ABB RobotStudio station: GoHolo_Simulation.rspag

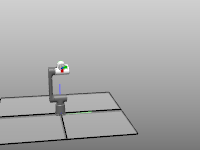
--- station ---
Station GoFa_Simulation (saved by RobotStudio 21.2.9526.0)
Controller GoFa
  mechanical unit ROB_1: CRB15000_5_95__01_2, 6 joints, base frame (0, 0, 0) mm
Layout (positions relative to the parent item):
  - CRB15000_5_95__01_2 [mechanism, from Robots\CRB15000_5_95__01.rslib] at (0, 0, 0) mm; joint values [0, 0, 0, 0, 0, 0] (rad or m)
Targets, tools, work objects and paths stored in the station and not in the controller backup, written as RAPID:
! task T_ROB1
MODULE module_MAIN
  CONST robtarget below:=[[500,0,500],[0,0,0,1],[0,0,0,0],[9E+09,9E+09,9E+09,9E+09,9E+09,9E+09]];
ENDMODULE

! task T_ROB1
MODULE MAINmodul
  PROC goHome()
    MoveJ pHome,v1000,fine,tool0\WObj:=wobj0;
  ENDPROC
ENDMODULE

! task T_ROB1
MODULE module_EGM
  PERS tooldata tEGM:=[TRUE,[[0,0,0],[1,0,0,0]],[0.001,[0,0,0.001],[1,0,0,0],0,0,0]];
  PROC EGM_Setup_UdpUC_Val()
    init_Val;
  ENDPROC
ENDMODULE

! task T_ROB1
MODULE EGM_Guidance
  PERS robtarget Target_10:=[[455.426,100,685.001],[0.5,-0.000000018,0.866025,0.000000059],[0,-1,0,0],[9E+09,9E+09,9E+09,9E+09,9E+09,9E+09]];
  PROC move()
    SingArea \LockAxis4;
  ENDPROC
  PROC EGM_UdpUC_VAL_Tool()
    EGM_Setup_UdpUC_Val;
    move;
    WaitTime 60;
    MoveJ Target_10,v100,fine,tEGM\WObj:=wobj0;
  ENDPROC
ENDMODULE

! task T_ROB1
MODULE module_WIZARD
  PERS robtarget Location3:=[[-0.096782632,525.209777832,576.337219238],[0.606442034,-0.534831524,0.457359105,0.370143116],[-1,-1,1,4],[-170.223126067,9E+09,9E+09,9E+09,9E+09,9E+09]];
  CONST jointtarget j00:=[[0,0,0,0,0,0],[0,0,0,0,0,0]];
  CONST jointtarget j90:=[[90,0,0,0,0,0],[0,0,0,0,0,0]];
  CONST jointtarget j80:=[[0,0,80,0,0,0],[0,0,0,0,0,0]];
  CONST jointtarget j20:=[[20,20,20,20,20,20],[0,0,0,0,0,0]];
  CONST jointtarget j30:=[[30,30,30,30,30,30],[0,0,0,0,0,0]];
  CONST jointtarget j30neg:=[[-30,-30,-30,-30,-30,-30],[0,0,0,0,0,0]];
  CONST jointtarget j90neg:=[[-90,0,0,0,0,0],[0,0,0,0,0,0]];
ENDMODULE

! task T_ROB1
MODULE Module1
  CONST robtarget Target_20:=[[571,0,899],[0.707106781,0,0.707106781,0],[0,-1,0,0],[9E+09,9E+09,9E+09,9E+09,9E+09,9E+09]];
ENDMODULE


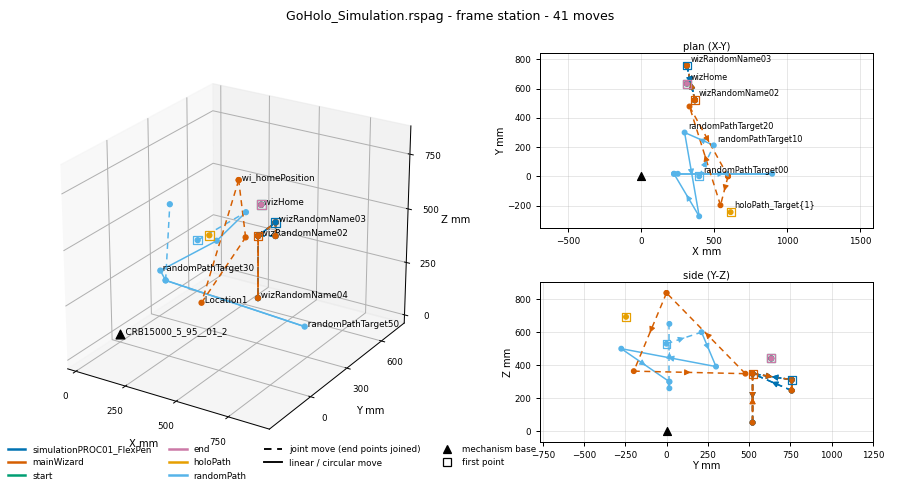
[picture p0: tool path of GoHolo_Simulation.rspag in frame station, 41 of 47 moves have a stored position in this frame; points joined in program order, loops and branches not executed]
--- Backups/GoFa/RAPID/TASK2/PROGMOD/module_MAIN.modx ---
MODULE module_MAIN
!
!       ---------------------------------
!                   GoHolo
!       ---------------------------------
!
!       Copyright (C)   2021 Jakob Hörbst
!       author:         Jakob Hörbst
!       email:          jakob@hoerbst.net
!       year:           2021
!

PROC main()
    mainGoHolo; ! hola die Waldfee
ENDPROC
ENDMODULE

--- Backups/GoFa/RAPID/TASK2/PROGMOD/module_WIZARD.modx ---
MODULE module_WIZARD
!
!       ---------------------------------
!                   GoHolo
!       ---------------------------------
!
!       Copyright (C)   2021 Jakob Hörbst
!       author:         Jakob Hörbst
!       email:          jakob@hoerbst.net
!       year:           2021
!

PERS robtarget wizHome:=[[316.17333984375, 634.73046875, 440.990356445313], [0.0026820998173207, 0.00783746875822544, 0.999948501586914, 0.00585808232426643], [0, 0, 0, 0], [9000000000, 9000000000, 9000000000, 9000000000, 9000000000, 9000000000]];
PERS robtarget wizRandomName02:=[[370.495269775391, 521.374877929688, 348.593353271484], [0.00379902473650873, 0.701789557933807, 0.712373673915863, -0.000882733904290944], [0, -1, 1, 0], [9000000000, 9000000000, 9000000000, 9000000000, 9000000000, 9000000000]];
PERS robtarget wizRandomName04:=[[370.480529785156, 521.381530761719, 51.8949508666992], [0.00380251440219581, 0.708827674388885, 0.705370903015137, -0.000862757791765034], [0, -1, 1, 0], [9000000000, 9000000000, 9000000000, 9000000000, 9000000000, 9000000000]];
PERS robtarget wizRandomName03:=[[314.93212890625, 758.710083007813, 311.827056884766], [0.00269204052165151, 0.00783240702003241, 0.999948382377625, 0.00589012308046222], [0, -1, 0, 0], [9000000000, 9000000000, 9000000000, 9000000000, 9000000000, 9000000000]];
PERS robtarget wizRandomName01:=[[314.909301757813, 758.708068847656, 246.256469726563], [0.00268639274872839, 0.00781508535146713, 0.999948561191559, 0.00588054535910487], [0, -1, 0, 0], [9000000000, 9000000000, 9000000000, 9000000000, 9000000000, 9000000000]];
PERS robtarget wizRandomName11:=[[370.495269775391, 521.374877929688, 348.593353271484], [0.00379902473650873, 0.701789557933807, 0.712373673915863, -0.000882733904290944], [0, -1, 1, 0], [9000000000, 9000000000, 9000000000, 9000000000, 9000000000, 9000000000]];
PERS robtarget wizRandomName13:=[[370.480529785156, 521.381530761719, 51.8949508666992], [0.00380251440219581, 0.708827674388885, 0.705370903015137, -0.000862757791765034], [0, -1, 1, 0], [9000000000, 9000000000, 9000000000, 9000000000, 9000000000, 9000000000]];
PERS robtarget wizRandomName14:=[[314.93212890625, 758.710083007813, 311.827056884766], [0.00269204052165151, 0.00783240702003241, 0.999948382377625, 0.00589012308046222], [0, -1, 0, 0], [9000000000, 9000000000, 9000000000, 9000000000, 9000000000, 9000000000]];
PERS robtarget wizRandomName12:=[[314.909301757813, 758.708068847656, 246.256469726563], [0.00268639274872839, 0.00781508535146713, 0.999948561191559, 0.00588054535910487], [0, -1, 0, 0], [9000000000, 9000000000, 9000000000, 9000000000, 9000000000, 9000000000]];
PROC simulationPROC01_FlexPendant()
    start;
    MoveJ wizRandomName03, v100, fine, tool0;
    MoveJ wizRandomName02, v100, fine, tool0;
    MoveJ wizRandomName03, v100, fine, tool0;
    MoveJ wizRandomName01, v100, fine, tool0;
    MoveJ wizRandomName02, v100, fine, tool0;
    MoveJ wizRandomName04, v100, fine, tool0;
    end;
ENDPROC
PROC mainWizard()
start;
MoveJ wizRandomName11, v100, fine, tool0;
MoveJ wizRandomName13, v100, fine, tool0;
MoveJ wizRandomName11, v100, fine, tool0;
MoveJ wizRandomName14, v100, fine, tool0;
MoveJ wizRandomName12, v100, fine, tool0;
MoveJ wizRandomName14, v100, fine, tool0;
end;
ENDPROC
PROC simulationPROC02_HoloLens2()
ENDPROC
PROC start()
    MoveJ wizHome, v200, fine, tool0;
ENDPROC
PROC end()
    MoveJ wizHome, v200, fine, tool0;
ENDPROC
ENDMODULE

--- Backups/GoFa/RAPID/TASK2/SYSMOD/module_EGM.sysx ---
MODULE module_EGM (SYSMODULE)

!
!       ---------------------------------
!                   GoHolo
!       ---------------------------------
!
!       Copyright (C)   2021 Jakob Hörbst
!       author:         Jakob Hörbst
!       email:          jakob@hoerbst.net
!       year:           2021
!

  !  PERS tooldata tEGM:=[TRUE,[[0,0,0],[1,0,0,0]],[0.001,[0,0,0.001],[1,0,0,0],0,0,0]];
    VAR egmident egmID1;
    VAR egmstate egmSt1;

    VAR egmident egmID_stream;
    VAR egmstate egmStStream;

    ! CONST egm_minmax egm_minmax_joint1:=[-0.1,0.1];
    ! Konvergenzkriterien AM EGM Seite 53
    CONST egm_minmax egm_minmax_lin1:=[-2,2]; ! in mm
    CONST egm_minmax egm_minmax_rot1:=[-2,2]; ! in °
    CONST pose posecor0:=[[0,0,0],[1,0,0,0]];


    ! was machen die beiden?!
    CONST pose posecor:=posecor0;![[1200,400,900], [0,0,1,0]];
    CONST pose posesens:=posecor0;![[12.3313,-0.108707,416.142],[0.903899,-0.00320735,0.427666,0.00765917]];


! GoHolo Setting kann verwendet werden für Fehler - Application Manuale EGM Seite 40

    PROC EGM_Init()
     !   tEGM:=CTool();

        EGMGetId egmID1;
        egmSt1:=EGMGetState(egmID1);
        IF egmSt1<=EGM_STATE_CONNECTED THEN
            EGMSetupUC ROB_1,egmID1,"GoHolo","UCdevice"\pose;
        ENDIF

        EGMActPose egmID1\StreamStart\Tool:=tool0\WObj:=wobj0,posecor,EGM_FRAME_WOBJ,posecor,EGM_FRAME_WOBJ
        \x:=egm_minmax_lin1\y:=egm_minmax_lin1\z:=egm_minmax_lin1\rx:=egm_minmax_rot1\ry:=egm_minmax_rot1\rz:=egm_minmax_rot1
        \MaxPosDeviation:=1000\MaxSpeedDeviation:=200; ! was 2x100

    ENDPROC

    PROC EGM_RunPose()

       ! SingArea \LockAxis4;
       ConfJ \Off;
       ConfL \Off;
        EGMRunPose egmID1,EGM_STOP_HOLD\x\y\z\Rx\Ry\Rz\RampInTime:=0.05;


         ERROR
            IF ERRNO=ERR_ROBLIMIT THEN
                TPWrite "Joint out of range error";
                !EGMReset egmID1;
            ELSEIF ERRNO=ERR_UDPUC_COMM THEN

                RETURN;
            ELSE
                STOP;
            ENDIF

    ENDPROC

    PROC EGM_Reset()
        EGMReset egmID_stream;
        EGMReset egmID1;
    ENDPROC

    PROC EGM_StreamStart()
        EGMGetId egmID_stream;
        egmStStream := EGMGetState(egmID_stream);
        IF egmStStream<=EGM_STATE_CONNECTED THEN
            EGMSetupUC ROB_1,egmID_stream,"default","UCstream"\Pose;
            EGMStreamStart egmID_stream;
        ENDIF
    ENDPROC

    PROC EGM_StreamStop()
        EGMGetId egmID_stream;
        egmStStream := EGMGetState(egmID_stream);
        IF egmStStream<=EGM_STATE_CONNECTED THEN
            EGMStreamStop egmID_stream;
        ENDIF
        EGMReset egmID_stream;
    ENDPROC

ENDMODULE

--- Backups/GoFa/RAPID/TASK2/SYSMOD/module_HOLOPATH.sysx ---
MODULE module_HOLOPATH (SYSMODULE)
!
!       ---------------------------------
!                   GoHolo
!       ---------------------------------
!
!       Copyright (C)   2021 Jakob Hörbst
!       author:         Jakob Hörbst
!       email:          jakob@hoerbst.net
!       year:           2021
!


    PERS jointtarget HP_startPos := [[0,0,0,0,0,0],[0,9E+09,9E+09,9E+09,9E+09,9E+09]];
    PERS robtarget holoPath_Target{10}:=[
        [[615.4, -245.4, 692.9],[-0.588, 0.063, -0.804, -0.061],[0, 0, 0, 0],[0,9E+9,9E+9,9E+9,9E+9,9E+9]],
        [[657.7, 202, 577.4],[-0.173, 0.192, -0.966, 0.02],[0, 0, 0, 0],[0,9E+9,9E+9,9E+9,9E+9,9E+9]],
        [[15.6, 547.8, 180.5],[0.357, -0.653, -0.59, -0.313],[0, 0, 0, 0],[0,9E+9,9E+9,9E+9,9E+9,9E+9]],
        [[573.6, 0, 689.9],[-0.707, 0, -0.707, 0],[0, 0, 0, 0],[0,9E+9,9E+9,9E+9,9E+9,9E+9]],
        [[0, 0, 0],[0, 1, 0, 0],[0, 0, 0, 1],[135,9E+9,9E+9,9E+9,9E+9,9E+9]],
        [[0, 0, 0],[0, 1, 0, 0],[0, 0, 0, 1],[135,9E+9,9E+9,9E+9,9E+9,9E+9]],
        [[0, 0, 0],[0, 1, 0, 0],[0, 0, 0, 1],[135,9E+9,9E+9,9E+9,9E+9,9E+9]],
        [[0, 0, 0],[0, 1, 0, 0],[0, 0, 0, 1],[135,9E+9,9E+9,9E+9,9E+9,9E+9]],
        [[0, 0, 0],[0, 1, 0, 0],[0, 0, 0, 1],[135,9E+9,9E+9,9E+9,9E+9,9E+9]],
        [[0, 0, 0],[0, 1, 0, 0],[0, 0, 0, 1],[135,9E+9,9E+9,9E+9,9E+9,9E+9]]
        ];
    PERS bool holoPath_TargetValid{10} := [
            TRUE,
            TRUE,
            TRUE,
            TRUE,
            TRUE,
            TRUE,
            TRUE,
            TRUE,
            TRUE,
            TRUE
        ];
    PERS bool validationComplete := TRUE;
    PERS bool simulationComplete := TRUE;

    VAR speeddata holoPath_Speed := v100;
    PERS num holoPath_TargetNumber := 2;
    PERS bool holoPathExecute := FALSE;

    PROC holoPath()
        VAR num duration; ! in s
        VAR clock chrono;

        MoveAbsJ HP_startPos, holoPath_Speed, fine, tool0\WObj:=wobj0;

        IF holoPathExecute THEN
            simulationComplete := FALSE;
            validationComplete := FALSE;

            ClkReset chrono;
            ClkStart chrono;

            ! check if the targets are valid and start movement if so
            IF checkTarget() THEN
                validationComplete := TRUE;
                ClkStop chrono;
                duration := ClkRead(chrono); ! in s

                !ConfJ\Off;
                IF holoPath_TargetNumber > 0 THEN
                    FOR holoPath_i FROM 1 TO holoPath_TargetNumber DO
                        IF holoPath_i = 1 THEN
                            MoveJ holoPath_Target{1}, holoPath_Speed, fine, tool0\WObj:=wobj0;
                        ELSE
                            MoveJ holoPath_Target{holoPath_i}, holoPath_Speed, fine, tool0\WObj:=wobj0;
                        ENDIF
                    ENDFOR
                ENDIF
                WaitRob \InPos;
                simulationComplete := TRUE;
                !ConfJ\On;
            ELSE
                 simulationComplete := FALSE;
                 validationComplete := TRUE;
            ENDIF

        ENDIF
        holoPathExecute := FALSE;
    ENDPROC

    ! checking if the targets from the MR-application are reachable in any configuration
    FUNC bool checkTarget()

        VAR robtarget rTar;
        VAR jointtarget jTar;
        VAR errnum errValidation;

        VAR num conf1;

        ! reset validation
        FOR i FROM 1 TO holoPath_TargetNumber DO holoPath_TargetValid{i} := FALSE; ENDFOR
        FOR i FROM holoPath_TargetNumber+1 TO 10 DO holoPath_TargetValid{i} := TRUE; ENDFOR

        ! cf1 axis1: from -2 to 1
        ! cf4 axis4: from -2 to 1
        ! cf6 axis6: from -2 to 2
        ! cfx config: from 0 to 7

            IF holoPath_TargetNumber > 0 THEN
                FOR checkTarget_i FROM 1 TO holoPath_TargetNumber DO
                    rTar := holoPath_Target{checkTarget_i};

                    FOR cf1 FROM -2 TO 1 DO
                        rTar.robconf.cf1 := cf1;

                        FOR cf4 FROM -2 TO 1 DO
                            rTar.robconf.cf4 := cf4;

                            FOR cf6 FROM -2 TO 1 DO
                                rTar.robconf.cf6 := cf6;

                                FOR cfx FROM 0 TO 7 DO
                                    rTar.robconf.cfx := cfx;

                                    jTar := CalcJointT(rTar, tool0 \ErrorNumber:=errValidation);

                                    IF NOT(errValidation = ERR_ROBLIMIT OR errValidation = ERR_OUTSIDE_REACH) THEN
                                        holoPath_TargetValid{checkTarget_i} := TRUE;
                                        GOTO tarValBreak; ! abort criteria
                                    ENDIF

                                ! END cfx
                                ENDFOR


                            ! END cf6
                            ENDFOR

                        ! END cf4
                        ENDFOR

                    ! END cf1
                    ENDFOR
                    tarValBreak:

                ! END list of targets
                ENDFOR

            ENDIF

        FOR i FROM 1 TO 10 DO
            IF holoPath_TargetValid{i} = FALSE THEN
                RETURN FALSE;
            ENDIF
        ENDFOR

        RETURN TRUE;

    ENDFUNC

ENDMODULE

--- Backups/GoFa/RAPID/TASK2/SYSMOD/module_MAIN_GOHOLO.sysx ---
MODULE module_MAIN_GOHOLO (SYSMODULE)
!
!       ---------------------------------
!                   GoHolo
!       ---------------------------------
!
!       Copyright (C)   2021 Jakob Hörbst
!       author:         Jakob Hörbst
!       email:          jakob@hoerbst.net
!       year:           2021
!


    ! INITIAL POSITIONS
    !CONST jointtarget pInitEGM          :=  [[0,0,25,0,-25,0], [0,0,0,0,0,0]];
    CONST jointtarget pInitEGM          :=  [[0,0,0,0,60,0], [0,0,0,0,0,0]];
    CONST jointtarget pInitStartup      :=  [[0,0,0,0,0,0], [0,0,0,0,0,0]];
    CONST robtarget pHome               :=  [[-200,100,300],[0,1,0,0],[2,0,0,0],[135,9E+09,9E+09,9E+09,9E+09,9E+09]];

    ! JOINT CONTROL
    PERS jointtarget jointControlTarget :=  [[0,0,0,0,0,0],[0,0,0,0,0,0]];
    VAR jointtarget jointControlTarDef  := [[0,0,0,0,0,0],[0,0,0,0,0,0]];
    PERS bool actJointControlTarget     :=  FALSE;

    ! COMANDS
    PERS num mode                       :=  0;
    VAR num modePrev;
    VAR num modePrevTerminate           :=  0;
    VAR bool bStartup                   :=  TRUE;
    VAR bool modeChanged                :=  FALSE;

    ! TERMINATING TARGET FOR EGM
    VAR robtarget tar;

    PERS bool startSimulation := FALSE;

    !!!!!!!!!!!!!!!!!!!!!!!!!!!!!!!!!!!!!!!!!!!!!!!!!!!!!!!!!!!!!!!!!!!!!!!!!!!!!!!!!!!!!!!!
    !!!!!!!!!!!!!!!!!!!!!!!!!!!!!!!!!!!!!!!!  MAIN  !!!!!!!!!!!!!!!!!!!!!!!!!!!!!!!!!!!!!!!!
    !!!!!!!!!!!!!!!!!!!!!!!!!!!!!!!!!!!!!!!!!!!!!!!!!!!!!!!!!!!!!!!!!!!!!!!!!!!!!!!!!!!!!!!!
    PROC mainGoHolo()

        ! Startup procedure
        IF bStartup THEN
            Startup;
            bStartup := FALSE;
        ENDIF

        ! Check if mode changed (externally)
        IF mode <> modePrevTerminate AND (mode >= 0 AND mode <= 5) THEN
            Modehandler;
        ENDIF

        ! RUN SELECTED MODE
        TEST mode
            CASE 0: ! DO NOTHING
!                MoveAbsJ pInitStartup, v100, fine, tool0;

            CASE 1: ! RANDOM PATH
                EGM_StreamStart;
                SingArea \Off;
                randomPath;

            CASE 2: ! EGM
                MoveAbsJ pInitEGM, v100, fine, tool0;
                EGM_Init;
                DeleteTrap;
                mode := 20;
            CASE 20:
                EGM_RunPose;

            CASE 3: ! JOINT CONTROL
                IF actJointControlTarget THEN
                    JointControl;
                    actJointControlTarget := FALSE;
                ENDIF

            CASE 4: ! HOLO PATHS
                SingArea \Off;
                holoPath;

            CASE 5: ! WIZARD SIMULATION
                mode := 50;
               ! STOP;
            CASE 50:
                IF startSimulation THEN
                    ConfJ \On;
                    ConfL \On;
                    mainWizard;
                    startSimulation := FALSE;
                    mode := 0;
                    ConfJ \Off;
                    ConfL \Off;

                ENDIF
        ENDTEST

    ENDPROC

    !
    !   STARTUP
    !
    PROC Startup()
        mode := 0;
        modePrevTerminate := -1; ! just any number to make a difference
        modeChanged := TRUE;
        !MotionSup \TuneValue:=50; ! default value

        holoPathExecute := FALSE;
        actJointControlTarget := FALSE;

        jointControlTarget := jointControlTarDef;

        EGM_StreamStart;

        ! INIT TRAP
        DeleteTrap;
        AddTrap;

        MoveAbsJ pInitStartup, v100, fine, tool0;
    ENDPROC

    !
    !   ModeHanlder
    !
    PROC Modehandler()
        ! If prev mode was EGM terminate EGM
        IF modePrevTerminate = 2 THEN
            SingArea \Off;
            tar := CRobT(\Tool:=tool0, \WObj:=wobj0);
                 MoveJ tar, v100, fine, tool0;
        ENDIF

        ! stop and reset EGM
        EGM_StreamStop;
        WaitTime 0.05;
        EGM_Reset;
        WaitTime 0.05;

        IF mode <> 2 THEN
            EGM_StreamStart;
            DeleteTrap;
            AddTrap;
        ENDIF

        modePrevTerminate := mode;
    ENDPROC

    !
    !   JOINT CONTROL
    !
    PROC JointControl()
        MoveAbsJ jointControlTarget, v200, z0, tool0;
    ENDPROC

    !
    ! TRAP (called when mode is changed)
    !
    PROC DeleteTrap()
        IDelete modePrev;
    ENDPROC

    PROC AddTrap()
        CONNECT modePrev WITH modeChangedTrap;
        IPers mode, modePrev;
    ENDPROC

    TRAP modeChangedTrap
        IF mode >= 0 AND mode <= 5 THEN
            !modeChanged := TRUE;
            ExitCycle;
        ENDIF
    ENDTRAP


ENDMODULE

--- Backups/GoFa/RAPID/TASK2/SYSMOD/module_RANDOMPATH.sysx ---
MODULE module_RANDOMPATH (SYSMODULE)
!
!       ---------------------------------
!                   GoHolo
!       ---------------------------------
!
!       Copyright (C)   2021 Jakob Hörbst
!       author:         Jakob Hörbst
!       email:          jakob@hoerbst.net
!       year:           2021
!


    ! RANDOM PATH
    CONST robtarget randomPathTarget00:=[[400,0,530],[0.5,0,0.866025404,0],[0,0,0,0],[9E+09,9E+09,9E+09,9E+09,9E+09,9E+09]];
    CONST robtarget randomPathTarget10:=[[500,212.17119565,600],[0.372760006,-0.5370996,0.745736898,0.128259412],[0,-1,-1,0],[9E+09,9E+09,9E+09,9E+09,9E+09,9E+09]];
    CONST robtarget randomPathTarget20:=[[300,300,391.552096279],[0.026136637,-0.60685633,0.794057513,-0.022692201],[0,-1,-1,0],[9E+09,9E+09,9E+09,9E+09,9E+09,9E+09]];
    CONST robtarget randomPathTarget30:=[[400,-274.159707825,500],[0.02613664,-0.606856313,0.794057525,-0.022692264],[-1,0,-2,0],[9E+09,9E+09,9E+09,9E+09,9E+09,9E+09]];
    CONST robtarget randomPathTarget40:=[[227.290100304,17.365610106,300],[0.026136653,-0.606856329,0.794057512,-0.022692262],[0,-1,-1,0],[9E+09,9E+09,9E+09,9E+09,9E+09,9E+09]];
    CONST robtarget randomPathTarget50:=[[900,17.365611158,259.858480384],[0.026136644,-0.60685631,0.794057527,-0.022692255],[0,-1,-1,0],[9E+09,9E+09,9E+09,9E+09,9E+09,9E+09]];
    CONST robtarget randomPathTarget60:=[[253.740697546,17.36560977,650.310810579],[0.607005214,0.022414458,0.027561649,0.793903406],[0,-1,1,1],[9E+09,9E+09,9E+09,9E+09,9E+09,9E+09]];

    !
    !   RANDOM PATH
    !
    PROC randomPath()
        VAR speeddata randomPath_Speed := v100;

        ConfJ \On;
        ConfL \On;
        MoveJ randomPathTarget00,randomPath_Speed,z100,tool0\WObj:=wobj0;
        MoveJ randomPathTarget10,randomPath_Speed,z100,tool0\WObj:=wobj0;
        MoveL randomPathTarget20,randomPath_Speed,z100,tool0\WObj:=wobj0;
        MoveL randomPathTarget30,randomPath_Speed,z100,tool0\WObj:=wobj0;
        MoveL randomPathTarget40,randomPath_Speed,z100,tool0\WObj:=wobj0;
        MoveL randomPathTarget50,randomPath_Speed,z100,tool0\WObj:=wobj0;
        MoveL randomPathTarget40,randomPath_Speed,z100,tool0\WObj:=wobj0;
        MoveJ randomPathTarget60,randomPath_Speed,z100,tool0\WObj:=wobj0;
    ENDPROC

ENDMODULE

--- Backups/GoFa/RAPID/TASK2/SYSMOD/Wizard_Params.sysx ---
MODULE Wizard_Params (SYSMODULE)
    !***************************************************************************
    !*                              Common parameters                          *
    !***************************************************************************
    ! Predefined common targets for user to use
    CONST jointtarget wi_jPosCalib:=[[0,0,0,0,30,0],[9E+9,9E+9,9E+9,9E+9,9E+9,9E+9]];

	PERS robtarget wi_homePosition:=[[597.47,0.00,837.78],[0.5,0,0.866025,0],[0,0,0,0],[9E+9,9E+9,9E+9,9E+9,9E+9,9E+9]];

    VAR errnum wi_errnum;

    PERS bool wi_bFirstLaunched:=FALSE;

    PERS num wi_asiMoveType:=0;

ENDMODULE

--- Backups/GoFa/RAPID/TASK3/PROGMOD/module_GETDATA.modx ---
MODULE module_GETDATA

    VAR num feedbackPosition{6};
    VAR num feedbackSpeed{6};
    VAR num feedbackTorque{6};
    VAR num feedbackExtTorque{6};

    VAR clock timer;
    VAR num duration;

    PROC main()
        GetData;
        WaitTime 0.015;
    ENDPROC

    PROC GetData()

        !torque := GetMotorTorque(2);
        FOR i FROM 1 TO 6 DO
            GetJointData\MechUnit:=ROB_1,i\position:=feedbackPosition{i}\speed:=feedbackSpeed{i}\torque:=feedbackTorque{i}\ExtTorque:=feedbackExtTorque{i};
        ENDFOR

        ClkStop timer;
        duration := ClkRead(timer)*1000;

        ClkReset timer;
        ClkStart timer;
    ENDPROC


ENDMODULE

--- Backups/GoFa/HOME/module_MAIN.modx ---
MODULE module_MAIN
PROC main()
    mainGoHolo; ! hola die Waldfee
ENDPROC
ENDMODULE

--- Backups/GoFa/HOME/module_WIZARD.modx ---
MODULE module_WIZARD
PERS robtarget wizHome:=[[316.17333984375, 634.73046875, 440.990356445313], [0.0026820998173207, 0.00783746875822544, 0.999948501586914, 0.00585808232426643], [0, 0, 0, 0], [9000000000, 9000000000, 9000000000, 9000000000, 9000000000, 9000000000]];
PERS robtarget wizRandomName02:=[[370.495269775391, 521.374877929688, 348.593353271484], [0.00379902473650873, 0.701789557933807, 0.712373673915863, -0.000882733904290944], [0, -1, 1, 0], [9000000000, 9000000000, 9000000000, 9000000000, 9000000000, 9000000000]];
PERS robtarget wizRandomName04:=[[370.480529785156, 521.381530761719, 51.8949508666992], [0.00380251440219581, 0.708827674388885, 0.705370903015137, -0.000862757791765034], [0, -1, 1, 0], [9000000000, 9000000000, 9000000000, 9000000000, 9000000000, 9000000000]];
PERS robtarget wizRandomName03:=[[314.93212890625, 758.710083007813, 311.827056884766], [0.00269204052165151, 0.00783240702003241, 0.999948382377625, 0.00589012308046222], [0, -1, 0, 0], [9000000000, 9000000000, 9000000000, 9000000000, 9000000000, 9000000000]];
PERS robtarget wizRandomName01:=[[314.909301757813, 758.708068847656, 246.256469726563], [0.00268639274872839, 0.00781508535146713, 0.999948561191559, 0.00588054535910487], [0, -1, 0, 0], [9000000000, 9000000000, 9000000000, 9000000000, 9000000000, 9000000000]];
PERS robtarget wizRandomName11:=[[370.495269775391, 521.374877929688, 348.593353271484], [0.00379902473650873, 0.701789557933807, 0.712373673915863, -0.000882733904290944], [0, -1, 1, 0], [9000000000, 9000000000, 9000000000, 9000000000, 9000000000, 9000000000]];
PERS robtarget wizRandomName13:=[[370.480529785156, 521.381530761719, 51.8949508666992], [0.00380251440219581, 0.708827674388885, 0.705370903015137, -0.000862757791765034], [0, -1, 1, 0], [9000000000, 9000000000, 9000000000, 9000000000, 9000000000, 9000000000]];
PERS robtarget wizRandomName14:=[[314.93212890625, 758.710083007813, 311.827056884766], [0.00269204052165151, 0.00783240702003241, 0.999948382377625, 0.00589012308046222], [0, -1, 0, 0], [9000000000, 9000000000, 9000000000, 9000000000, 9000000000, 9000000000]];
PERS robtarget wizRandomName12:=[[314.909301757813, 758.708068847656, 246.256469726563], [0.00268639274872839, 0.00781508535146713, 0.999948561191559, 0.00588054535910487], [0, -1, 0, 0], [9000000000, 9000000000, 9000000000, 9000000000, 9000000000, 9000000000]];
PROC simulationPROC01_FlexPendant()
    start;
    MoveJ wizRandomName03, v100, fine, tool0;
    MoveJ wizRandomName02, v100, fine, tool0;
    MoveJ wizRandomName03, v100, fine, tool0;
    MoveJ wizRandomName01, v100, fine, tool0;
    MoveJ wizRandomName02, v100, fine, tool0;
    MoveJ wizRandomName04, v100, fine, tool0;
    end;
ENDPROC
PROC mainWizard()
start;
MoveJ wizRandomName11, v100, fine, tool0;
MoveJ wizRandomName13, v100, fine, tool0;
MoveJ wizRandomName11, v100, fine, tool0;
MoveJ wizRandomName14, v100, fine, tool0;
MoveJ wizRandomName12, v100, fine, tool0;
MoveJ wizRandomName14, v100, fine, tool0;
end;
ENDPROC
PROC simulationPROC02_HoloLens2()
ENDPROC
PROC start()
    MoveJ wizHome, v200, fine, tool0;
ENDPROC
PROC end()
    MoveJ wizHome, v200, fine, tool0;
ENDPROC
ENDMODULE

--- Backups/GoFa/HOME/module_WIZARD123.modx ---
MODULE module_WIZARD
PERS robtarget Location1:=[[545.686218261719, -198.31755065918, 363.912017822266], [0.095397785305977, 0.127845048904419, 0.985680937767029, -0.054662574082613], [-1, -1, 0, 0], [9000000000, 9000000000, 9000000000, 9000000000, 9000000000, 9000000000]];
PERS robtarget Location2:=[[333.517272949219, 478.111175537109, 348.578552246094], [0.082118004560471, -0.467257678508759, 0.879561245441437, 0.0360402166843414], [0, -1, 0, 0], [9000000000, 9000000000, 9000000000, 9000000000, 9000000000, 9000000000]];
PROC mainWizard()
MoveJ wi_homePosition, v200, fine, tool0;
MoveJ Location1, v200, fine, tool0;
MoveJ Location2, v200, fine, tool0;
MoveJ wi_homePosition, v200, fine, tool0;
ENDPROC
ENDMODULE

--- Backups/GoFa/SYSPAR/EIO.cfg ---
EIO:CFG_1.0:7:0::

#CTRL_SIGNATURE:S+LYcqArLMmGZgqqjjGUBD/8e6ezfqGpXPR2BCTNCsk/WHzQTb5qC5zDA7HnBTpGYs4kTDiZqpucexzxOWDM2Q==

--- Backups/GoFa/SYSPAR/PROC.cfg ---
PROC:CFG_1.0:7:0::

#CTRL_SIGNATURE:I+y2QaV15gWtHGM+5Z4idi3NiusZu29hLyokxM3ohwogLM8MfydOTWOtI2G6szFitByh5svEYsXD7agPogo+dQ==
